TYPE "UDT_STATUS_PLANTA"
VERSION : 0.1
   STRUCT
      BRITADORES  : "UDT_STATUS_BRITADORES";
      TRANSPORTADORES  : "UDT_STATUS_TRANSPORTADORES";
      PENEIRAS  : "UDT_STATUS_PENEIRAS";
      CALHAS  : "UDT_STATUS_CALHAS";
      GLOBAL : Bool;
   END_STRUCT;

END_TYPE

